Staubli VAL3: check.pgx

program check()
begin
  while taskStatus("comunication")!=-1
    if taskStatus("comunication")>1
      // try to clear the buffer and resume
      clearBuffer(io:tcp_client)
      taskKill("comunication")
      wait(taskStatus("comunication")==-1)
      // create the task again from the beginning
      taskCreate "comunication",10,comunication()
    endIf
    delay(0)
  endWhile
end
